SUBAPPLICATION SubApp_Proximity_Sensor (* Subapplication Type *)
  (* Standard: 61499-2 *)
  (* Version 1.0, 2022-10-10, AK123957 *)
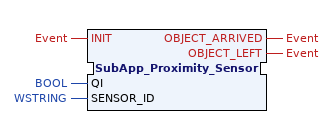
  EVENT_INPUT
    INIT;
  END_EVENT
  EVENT_OUTPUT
    OBJECT_ARRIVED;
    OBJECT_LEFT;
  END_EVENT
  VAR_INPUT
    QI : BOOL;
    SENSOR_ID : WSTRING;
  END_VAR
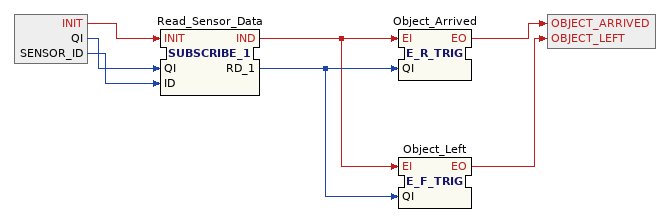
  FBS
    Object_Arrived : E_R_TRIG;
    Read_Sensor_Data : SUBSCRIBE_1;
    Object_Left : E_F_TRIG;
  END_FBS
  EVENT_CONNECTIONS
    Read_Sensor_Data.IND TO Object_Arrived.EI;
    Read_Sensor_Data.IND TO Object_Left.EI;
    INIT TO Read_Sensor_Data.INIT;
    Object_Arrived.EO TO OBJECT_ARRIVED;
    Object_Left.EO TO OBJECT_LEFT;
  END_CONNECTIONS
  DATA_CONNECTIONS
    Read_Sensor_Data.RD_1 TO Object_Arrived.QI;
    Read_Sensor_Data.RD_1 TO Object_Left.QI;
    QI TO Read_Sensor_Data.QI;
    SENSOR_ID TO Read_Sensor_Data.ID;
  END_CONNECTIONS
END_SUBAPPLICATION
